PROGRAM prgModeRows
VAR
	
ModeRow1:FB_HMI_Control_NoGroupRef;
ModeRow2:FB_HMI_Control_NoGroupRef;
ModeRow3:FB_HMI_Control_NoGroupRef;
ModeRow4:FB_HMI_Control_NoGroupRef;
ModeRow5:FB_HMI_Control_NoGroupRef;
ModeRow6:FB_HMI_Control_NoGroupRef;
ModeRow7:FB_HMI_Control_NoGroupRef;
ModeRow8:FB_HMI_Control_NoGroupRef;
ModeRow9:FB_HMI_Control_NoGroupRef;

ModeRowsStn: typeStation;
	tNumRows: UINT;
END_VAR

VAR_INPUT
	MotionRowLocation: typeMotionRow;
END_VAR

//theme:VNPKlVq0z2Y

//zero indexing code
tNumRows := 0;

//clear HMI row for manual insertion
gModeAlternate.gModeRows.gMotionRow1.IndexLocation := 0;
gModeAlternate.gModeRows.gMotionRow2.IndexLocation := 20;
gModeAlternate.gModeRows.gMotionRow3.IndexLocation := 40;
gModeAlternate.gModeRows.gMotionRow4.IndexLocation := 60;
gModeAlternate.gModeRows.gMotionRow5.IndexLocation := 80;
gModeAlternate.gModeRows.gMotionRow6.IndexLocation := 100;
gModeAlternate.gModeRows.gMotionRow7.IndexLocation := 120;
gModeAlternate.gModeRows.gMotionRow8.IndexLocation := 140;
gModeAlternate.gModeRows.gMotionRow9.IndexLocation := 160;

//call the rows
actcallRows();

ACTION actCallRows:
//theme:ETfiUYij5UE
//hard code location and address for special case of alternate motion row use for mode


//motion row 1, Power ON/OFF
ModeRow1	(	iStationNumber		:=1,
				iRowNumber			:=1,
				iAdvanceLimit		:=Mc_Global.PowerOnFdbk,
				iReturnLimit		:=NOT Mc_Global.PowerOnFdbk,
				iAdvanceCoil		:=gModeAlternate.gModeButtons.gMotionRow1btn.btnAdvance,
				iReturnCoil			:=gModeAlternate.gModeButtons.gMotionRow1btn.btnReturn,
				iAdvanceTime		:=,
				iReturnTime			:=,
				iAdvanceInterlock	:=,
				iReturnInterlock	:=,
				iAdvancePrompt		:=,
				iReturnPrompt		:=,
				iConfig				:=RowConfig.FullRowNoVal,
				iAdvanceNumber		:=0,
				iReturnNumber		:=0,
				iUnits				:='',
				iPosn				:='',
				NumRows				:=tNumRows,
				MotionRowLocation	:=gModeAlternate.gModeRows.gMotionRow1,
				MotionRowBtnLocation:=gModeAlternate.gModeButtons.gMotionRow1btn
				);

//manually set row number for textlist offset				
gModeAlternate.gModeRows.gMotionRow1.IndexLocation := gModeAlternate.gModeRows.gMotionRow1.IndexLocation + 10000;			


//motion row 2, Auto / Manual
ModeRow2	(	iStationNumber		:=1,
				iRowNumber			:=2,
				iAdvanceLimit		:=gHMIButtons.btnFdbk.btn00Fdbk,
				iReturnLimit		:=gHMIButtons.btnFdbk.btn01Fdbk,
				iAdvanceCoil		:=gModeAlternate.gModeButtons.gMotionRow2btn.btnAdvance,
				iReturnCoil			:=gModeAlternate.gModeButtons.gMotionRow2btn.btnReturn,
				iAdvanceTime		:=,
				iReturnTime			:=,
				iAdvanceInterlock	:=,
				iReturnInterlock	:=,
				iAdvancePrompt		:=,
				iReturnPrompt		:=,
				iConfig				:=RowConfig.FullRowNoVal,
				iAdvanceNumber		:=0,
				iReturnNumber		:=0,
				iUnits				:='',
				iPosn				:='',
				NumRows				:=tNumRows,
				MotionRowLocation	:=gModeAlternate.gModeRows.gMotionRow2,
				MotionRowBtnLocation:=gModeAlternate.gModeButtons.gMotionRow2btn
				);
				
				
//manually set row number for textlist offset				
gModeAlternate.gModeRows.gMotionRow2.IndexLocation := gModeAlternate.gModeRows.gMotionRow2.IndexLocation + 10000;			


//motion row 3, cycle cont / single
ModeRow3	(	iStationNumber		:=1,
				iRowNumber			:=3,
				iAdvanceLimit		:=gHMIButtons.btnFdbk.btn10Fdbk,
				iReturnLimit		:=gHMIButtons.btnFdbk.btn13Fdbk,
				iAdvanceCoil		:=gModeAlternate.gModeButtons.gMotionRow3btn.btnAdvance,
				iReturnCoil			:=gModeAlternate.gModeButtons.gMotionRow3btn.btnReturn,
				iAdvanceTime		:=,
				iReturnTime			:=,
				iAdvanceInterlock	:=,
				iReturnInterlock	:=,
				iAdvancePrompt		:=,
				iReturnPrompt		:=,
				iConfig				:=RowConfig.FullRowNoVal,
				iAdvanceNumber		:=0,
				iReturnNumber		:=0,
				iUnits				:='',
				iPosn				:='',
				NumRows				:=tNumRows,
				MotionRowLocation	:=gModeAlternate.gModeRows.gMotionRow3,
				MotionRowBtnLocation:=gModeAlternate.gModeButtons.gMotionRow3btn
				);
				
//manually set row number for textlist offset				
gModeAlternate.gModeRows.gMotionRow3.IndexLocation := gModeAlternate.gModeRows.gMotionRow3.IndexLocation + 10000;			


//motion row 4, cycle start / stop
ModeRow4	(	iStationNumber		:=1,
				iRowNumber			:=4,
				iAdvanceLimit		:=gHMIButtons.btnFdbk.btnAutoCyclingFdbk,
				iReturnLimit		:=NOT gHMIButtons.btnFdbk.btnAutoCyclingFdbk,
				iAdvanceCoil		:=gModeAlternate.gModeButtons.gMotionRow4btn.btnAdvance,
				iReturnCoil			:=gModeAlternate.gModeButtons.gMotionRow4btn.btnReturn,
				iAdvanceTime		:=,
				iReturnTime			:=,
				iAdvanceInterlock	:=,
				iReturnInterlock	:=,
				iAdvancePrompt		:=,
				iReturnPrompt		:=,
				iConfig				:=RowConfig.FullRowNoVal,
				iAdvanceNumber		:=0,
				iReturnNumber		:=0,
				iUnits				:='',
				iPosn				:='',
				NumRows				:=tNumRows,
				MotionRowLocation	:=gModeAlternate.gModeRows.gMotionRow4,
				MotionRowBtnLocation:=gModeAlternate.gModeButtons.gMotionRow4btn
				);
				
//manually set row number for textlist offset				
gModeAlternate.gModeRows.gMotionRow4.IndexLocation := gModeAlternate.gModeRows.gMotionRow4.IndexLocation + 10000;			

//motion row 5, return home
ModeRow5	(	iStationNumber		:=1,
				iRowNumber			:=5,
				iAdvanceLimit		:=gHMIData.hmiHeader.homestate = 2,
				iReturnLimit		:=gHMIData.hmiHeader.homestate <> 2,
				iAdvanceCoil		:=gModeAlternate.gModeButtons.gMotionRow5btn.btnAdvance,
				iReturnCoil			:=gModeAlternate.gModeButtons.gMotionRow5btn.btnReturn,
				iAdvanceTime		:=,
				iReturnTime			:=,
				iAdvanceInterlock	:=,
				iReturnInterlock	:=,
				iAdvancePrompt		:=,
				iReturnPrompt		:=,
				iConfig				:=RowConfig.OnlyRightNoVal,
				iAdvanceNumber		:=0,
				iReturnNumber		:=0,
				iUnits				:='',
				iPosn				:='',
				NumRows				:=tNumRows,
				MotionRowLocation	:=gModeAlternate.gModeRows.gMotionRow5,
				MotionRowBtnLocation:=gModeAlternate.gModeButtons.gMotionRow5btn
				);
				
//manually set row number for textlist offset				
gModeAlternate.gModeRows.gMotionRow5.IndexLocation := gModeAlternate.gModeRows.gMotionRow5.IndexLocation + 10000;			

//motion row 6, spare
ModeRow6	(	iStationNumber		:=1,
				iRowNumber			:=6,
				iAdvanceLimit		:=FALSE,
				iReturnLimit		:=FALSE,
				iAdvanceCoil		:=gModeAlternate.gModeButtons.gMotionRow6btn.btnAdvance,
				iReturnCoil			:=gModeAlternate.gModeButtons.gMotionRow6btn.btnReturn,
				iAdvanceTime		:=,
				iReturnTime			:=,
				iAdvanceInterlock	:=,
				iReturnInterlock	:=,
				iAdvancePrompt		:=,
				iReturnPrompt		:=,
				iConfig				:=RowConfig.HideAll,
				iAdvanceNumber		:=0,
				iReturnNumber		:=0,
				iUnits				:='',
				iPosn				:='',
				NumRows				:=tNumRows,
				MotionRowLocation	:=gModeAlternate.gModeRows.gMotionRow6,
				MotionRowBtnLocation:=gModeAlternate.gModeButtons.gMotionRow6btn
				);
				
//manually set row number for textlist offset				
gModeAlternate.gModeRows.gMotionRow6.IndexLocation := gModeAlternate.gModeRows.gMotionRow6.IndexLocation + 10000;			

//motion row 7, spare
ModeRow7	(	iStationNumber		:=1,
				iRowNumber			:=7,
				iAdvanceLimit		:=FALSE,
				iReturnLimit		:=FALSE,
				iAdvanceCoil		:=gModeAlternate.gModeButtons.gMotionRow7btn.btnAdvance,
				iReturnCoil			:=gModeAlternate.gModeButtons.gMotionRow7btn.btnReturn,
				iAdvanceTime		:=,
				iReturnTime			:=,
				iAdvanceInterlock	:=,
				iReturnInterlock	:=,
				iAdvancePrompt		:=,
				iReturnPrompt		:=,
				iConfig				:=RowConfig.HideAll,
				iAdvanceNumber		:=0,
				iReturnNumber		:=0,
				iUnits				:='',
				iPosn				:='',
				NumRows				:=tNumRows,
				MotionRowLocation	:=gModeAlternate.gModeRows.gMotionRow7,
				MotionRowBtnLocation:=gModeAlternate.gModeButtons.gMotionRow7btn
				);

//manually set row number for textlist offset				
gModeAlternate.gModeRows.gMotionRow7.IndexLocation := gModeAlternate.gModeRows.gMotionRow7.IndexLocation + 10000;			
				
//motion row 8, gate lock, return only
ModeRow8	(	iStationNumber		:=1,
				iRowNumber			:=8,
				iAdvanceLimit		:=FALSE,
				iReturnLimit		:=gHMIButtons.btnFdbk.btn22Fdbk,
				iAdvanceCoil		:=gModeAlternate.gModeButtons.gMotionRow8btn.btnAdvance,
				iReturnCoil			:=gModeAlternate.gModeButtons.gMotionRow8btn.btnReturn,
				iAdvanceTime		:=,
				iReturnTime			:=,
				iAdvanceInterlock	:=,
				iReturnInterlock	:=,
				iAdvancePrompt		:=,
				iReturnPrompt		:=,
				iConfig				:=RowConfig.OnlyRightNoVal,
				iAdvanceNumber		:=0,
				iReturnNumber		:=0,
				iUnits				:='',
				iPosn				:='',
				NumRows				:=tNumRows,
				MotionRowLocation	:=gModeAlternate.gModeRows.gMotionRow8,
				MotionRowBtnLocation:=gModeAlternate.gModeButtons.gMotionRow8btn
				);
				
//manually set row number for textlist offset				
gModeAlternate.gModeRows.gMotionRow8.IndexLocation := gModeAlternate.gModeRows.gMotionRow8.IndexLocation + 10000;			

//motion row 9, gate unlocks
ModeRow9	(	iStationNumber		:=1,
				iRowNumber			:=9,
				iAdvanceLimit		:=gHMIButtons.btnFdbk.btn20Fdbk,
				iReturnLimit		:=gHMIButtons.btnFdbk.btn21Fdbk,
				iAdvanceCoil		:=gModeAlternate.gModeButtons.gMotionRow9btn.btnAdvance,
				iReturnCoil			:=gModeAlternate.gModeButtons.gMotionRow9btn.btnReturn,
				iAdvanceTime		:=,
				iReturnTime			:=,
				iAdvanceInterlock	:=,
				iReturnInterlock	:=,
				iAdvancePrompt		:=,
				iReturnPrompt		:=,
				iConfig				:=RowConfig.FullRowNoVal,
				iAdvanceNumber		:=0,
				iReturnNumber		:=0,
				iUnits				:='',
				iPosn				:='',
				NumRows				:=tNumRows,
				MotionRowLocation	:=gModeAlternate.gModeRows.gMotionRow9,
				MotionRowBtnLocation:=gModeAlternate.gModeButtons.gMotionRow9btn
				);
				
//manually set row number for textlist offset				
gModeAlternate.gModeRows.gMotionRow9.IndexLocation := gModeAlternate.gModeRows.gMotionRow9.IndexLocation + 10000;
END_ACTION

END_PROGRAM

(* stored: Version 1.1.0.1, ProductVersion 3.1.4024.12
   POU prgModeRows: Id {767b4522-f0b4-4e13-b8aa-2d8f01ac42f8}, SpecialFunc None
   Action actCallRows: Id {131fe314-d854-446b-a3e7-9a871f15e3fe} *)
